// TIA Portal V20 export
DATA_BLOCK "FONCTION_DB_1"   // DB3
// stored: InstanceOfName Ely_2.FONCTION, InstanceOfType FB, Namespace Ely_2
"Ely_2.FONCTION"
BEGIN
END_DATA_BLOCK
